{attribute 'qualified_only'}
VAR_GLOBAL
	// Pitch Mechanism:
	{attribute 'TcLinkTo' := '.diEncCnt:=TIIB[EL5042_M1K4_PitchBender]^FB Inputs Channel 1^Position'}
	M1K4_Pitch : HOMS_PitchMechanism := (ReqPosLimHi := 275,
		                                 ReqPosLimLo := -25,
		                                 diEncPosLimHi := 10149192,
		                                 diEncPosLimLo := 10047105);
END_VAR

(* stored: Version 1.1.0.1, ProductVersion 3.1.4022.18
   GVL GVL_M1K4: Id {2074b16f-0d4c-4051-96e9-b5e1650ca1c7} *)
